// TIA Portal V19 export
TYPE "LEXCHANGETRAY_typeScanner_status"
// stored: Access Published
   STRUCT
      done : Bool;
      error { S7_SetPoint := 'True'} : Bool;
      ok : Bool;
      execute : Bool;
      cmdStep : Int;
   END_STRUCT;
END_TYPE
